(* CoDeSys 2.3 export: MNG_APPLICATION_INPUTS_32BIT.EXP *)

(* Data type *)
(*                                                                            *)

TYPE MNG_APPLICATION_INPUTS_32BIT :
STRUCT
    NumSignals                    : INT     := 5         ;
    CAR01_AXIS                    : REAL    := 0.0; (* Physics://physics/PCC/ALL/CAR?KinAxis *)
    CAR01_ACT_SPD                 : REAL    := 0.0; (* Physics://physics/PCC/ALL/CAR?KinSpeed *)
    CAR01_RCHD                    : BOOL    := 0; (* Physics://physics/PCC/ALL/CAR?KinReached *)
    pallet01_ButtonPress          : BOOL    := 0; (* /CAR/Platform/Fork/fork01/fork02/pallet?ButtonPress *)
    rectangular_tube_101_ButtonPre: BOOL    := 0; (* ics/PCC/ALL/CAR/Body/rectangular tube 1?ButtonPress *)
END_STRUCT
END_TYPE
